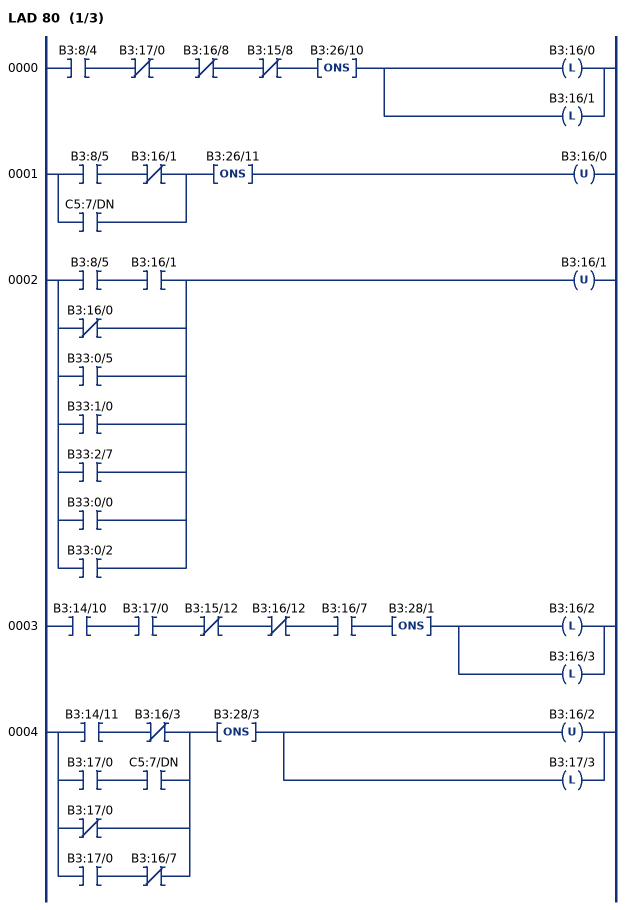
% Rung: 0 %
SOR XIC B3:8/4 XIO B3:17/0 XIO B3:16/8 XIO B3:15/8 OSR B3:26/10 BST OTL B3:16/0 NXB OTL B3:16/1 BND EOR
% Rung: 1 %
SOR BST XIC B3:8/5 XIO B3:16/1 NXB XIC C5:7/DN BND OSR B3:26/11 OTU B3:16/0 EOR
% Rung: 2 %
SOR BST XIC B3:8/5 XIC B3:16/1 NXB XIO B3:16/0 NXB XIC B33:0/5 NXB XIC B33:1/0 NXB XIC B33:2/7 NXB XIC B33:0/0 NXB XIC B33:0/2 BND OTU B3:16/1 EOR
% Rung: 3 %
SOR XIC B3:14/10 XIC B3:17/0 XIO B3:15/12 XIO B3:16/12 XIC B3:16/7 OSR B3:28/1 BST OTL B3:16/2 NXB OTL B3:16/3 BND EOR
% Rung: 4 %
SOR BST XIC B3:14/11 XIO B3:16/3 NXB XIC B3:17/0 XIC C5:7/DN NXB XIO B3:17/0 NXB XIC B3:17/0 XIO B3:16/7 BND OSR B3:28/3 BST OTU B3:16/2 NXB OTL B3:17/3 BND EOR

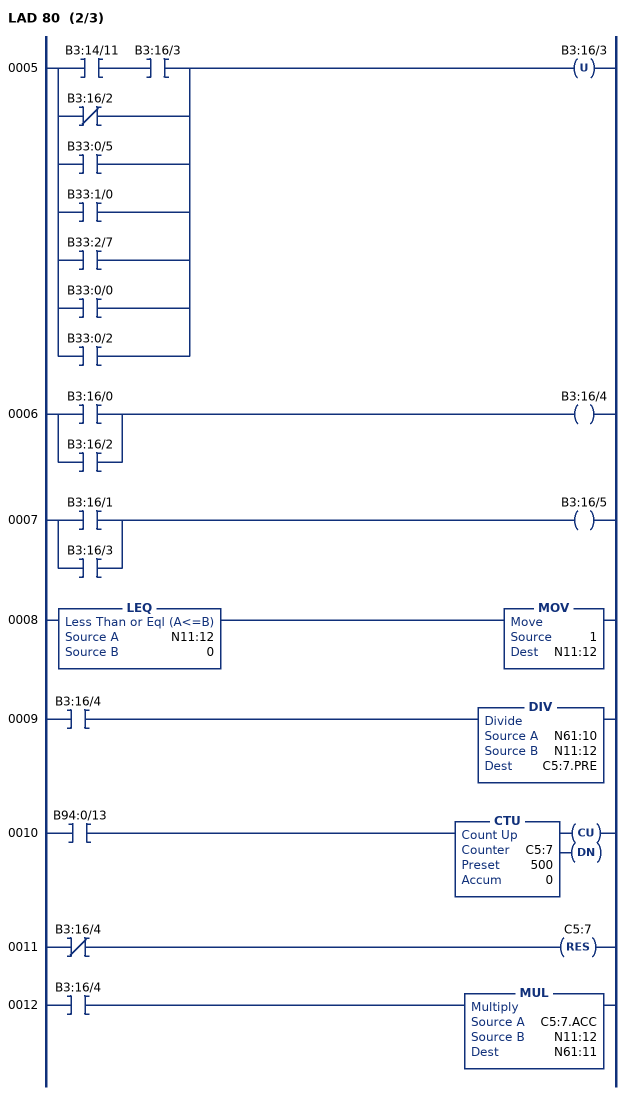
% Rung: 5 %
SOR BST XIC B3:14/11 XIC B3:16/3 NXB XIO B3:16/2 NXB XIC B33:0/5 NXB XIC B33:1/0 NXB XIC B33:2/7 NXB XIC B33:0/0 NXB XIC B33:0/2 BND OTU B3:16/3 EOR
% Rung: 6 %
SOR BST XIC B3:16/0 NXB XIC B3:16/2 BND OTE B3:16/4 EOR
% Rung: 7 %
SOR BST XIC B3:16/1 NXB XIC B3:16/3 BND OTE B3:16/5 EOR
% Rung: 8 %
SOR LEQ N11:12 0 MOV 1 N11:12 EOR
% Rung: 9 %
SOR XIC B3:16/4 DIV N61:10 N11:12 C5:7.PRE EOR
% Rung: 10 %
SOR XIC B94:0/13 CTU C5:7 500 0 EOR
% Rung: 11 %
SOR XIO B3:16/4 RES C5:7 EOR
% Rung: 12 %
SOR XIC B3:16/4 MUL C5:7.ACC N11:12 N61:11 EOR

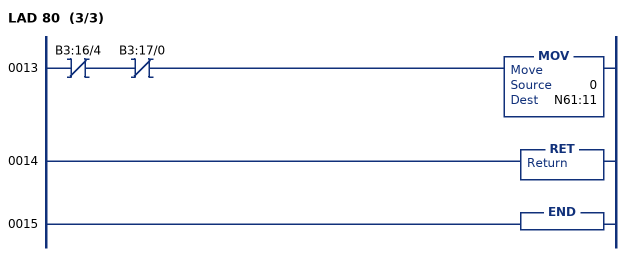
% Rung: 13 %
SOR XIO B3:16/4 XIO B3:17/0 MOV 0 N61:11 EOR
% Rung: 14 %
SOR RET EOR
% Rung: 15 %
SOR END EOR

LADDER 85
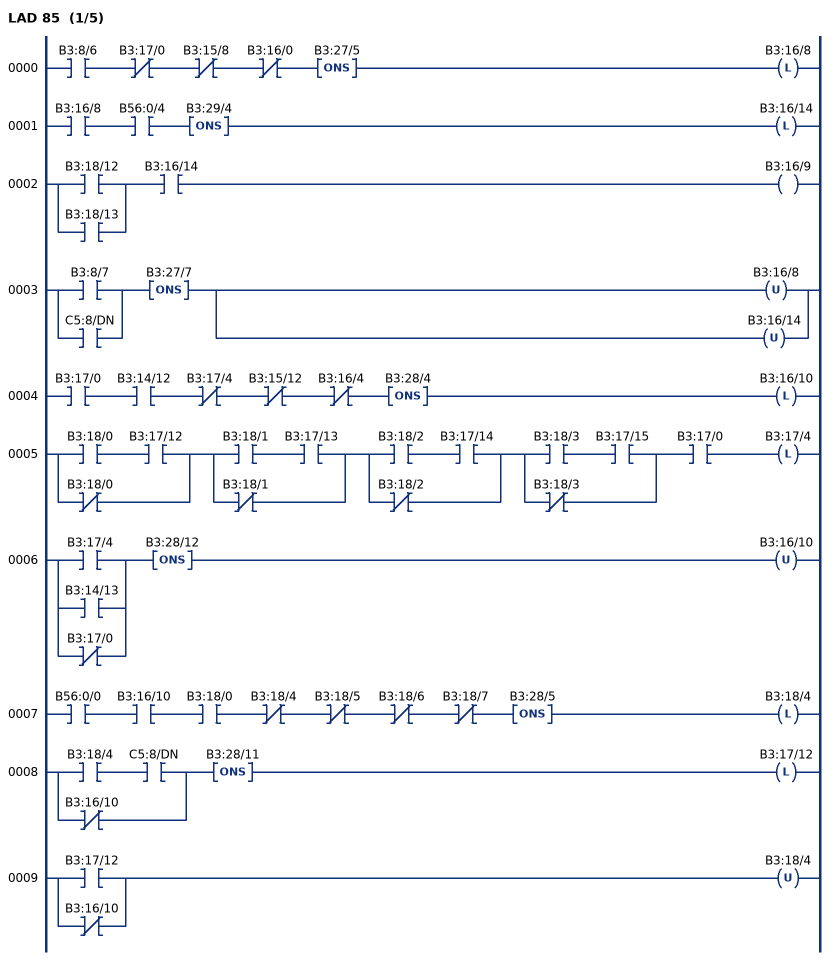
% Rung: 0 %
SOR XIC B3:8/6 XIO B3:17/0 XIO B3:15/8 XIO B3:16/0 OSR B3:27/5 OTL B3:16/8 EOR
% Rung: 1 %
SOR XIC B3:16/8 XIC B56:0/4 OSR B3:29/4 OTL B3:16/14 EOR
% Rung: 2 %
SOR BST XIC B3:18/12 NXB XIC B3:18/13 BND XIC B3:16/14 OTE B3:16/9 EOR
% Rung: 3 %
SOR BST XIC B3:8/7 NXB XIC C5:8/DN BND OSR B3:27/7 BST OTU B3:16/8 NXB OTU B3:16/14 BND EOR
% Rung: 4 %
SOR XIC B3:17/0 XIC B3:14/12 XIO B3:17/4 XIO B3:15/12 XIO B3:16/4 OSR B3:28/4 OTL B3:16/10 EOR
% Rung: 5 %
SOR BST XIC B3:18/0 XIC B3:17/12 NXB XIO B3:18/0 BND BST XIC B3:18/1 XIC B3:17/13 NXB XIO B3:18/1 BND BST XIC B3:18/2 XIC B3:17/14 NXB XIO B3:18/2 BND BST XIC B3:18/3 XIC B3:17/15 NXB XIO B3:18/3 BND XIC B3:17/0 OTL B3:17/4 EOR
% Rung: 6 %
SOR BST XIC B3:17/4 NXB XIC B3:14/13 NXB XIO B3:17/0 BND OSR B3:28/12 OTU B3:16/10 EOR
% Rung: 7 %
SOR XIC B56:0/0 XIC B3:16/10 XIC B3:18/0 XIO B3:18/4 XIO B3:18/5 XIO B3:18/6 XIO B3:18/7 OSR B3:28/5 OTL B3:18/4 EOR
% Rung: 8 %
SOR BST XIC B3:18/4 XIC C5:8/DN NXB XIO B3:16/10 BND OSR B3:28/11 OTL B3:17/12 EOR
% Rung: 9 %
SOR BST XIC B3:17/12 NXB XIO B3:16/10 BND OTU B3:18/4 EOR

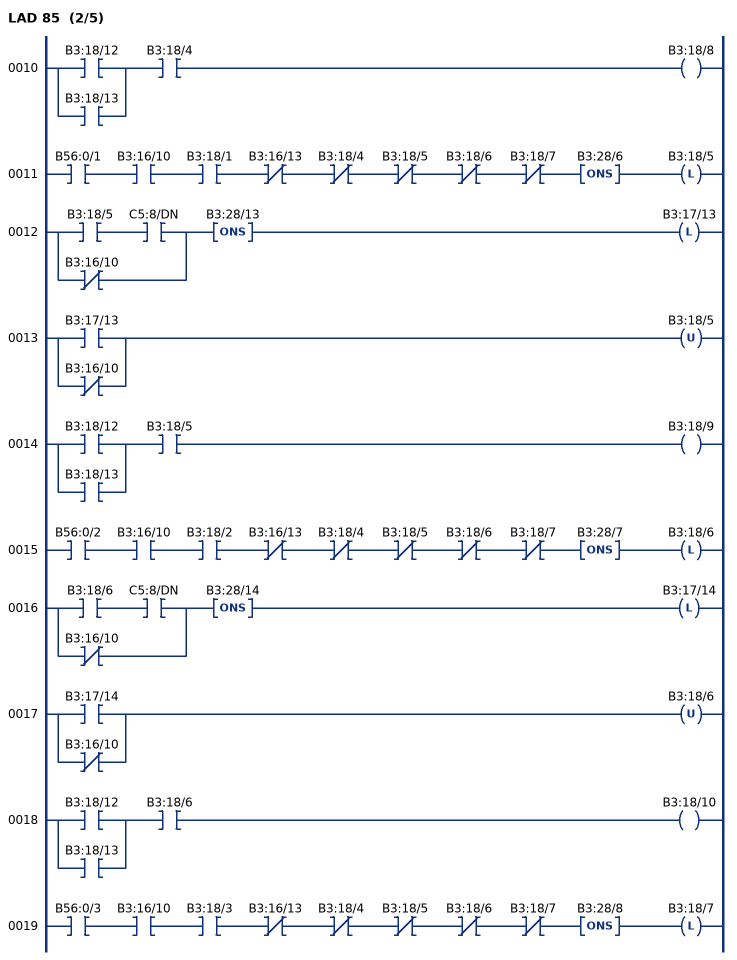
% Rung: 10 %
SOR BST XIC B3:18/12 NXB XIC B3:18/13 BND XIC B3:18/4 OTE B3:18/8 EOR
% Rung: 11 %
SOR XIC B56:0/1 XIC B3:16/10 XIC B3:18/1 XIO B3:16/13 XIO B3:18/4 XIO B3:18/5 XIO B3:18/6 XIO B3:18/7 OSR B3:28/6 OTL B3:18/5 EOR
% Rung: 12 %
SOR BST XIC B3:18/5 XIC C5:8/DN NXB XIO B3:16/10 BND OSR B3:28/13 OTL B3:17/13 EOR
% Rung: 13 %
SOR BST XIC B3:17/13 NXB XIO B3:16/10 BND OTU B3:18/5 EOR
% Rung: 14 %
SOR BST XIC B3:18/12 NXB XIC B3:18/13 BND XIC B3:18/5 OTE B3:18/9 EOR
% Rung: 15 %
SOR XIC B56:0/2 XIC B3:16/10 XIC B3:18/2 XIO B3:16/13 XIO B3:18/4 XIO B3:18/5 XIO B3:18/6 XIO B3:18/7 OSR B3:28/7 OTL B3:18/6 EOR
% Rung: 16 %
SOR BST XIC B3:18/6 XIC C5:8/DN NXB XIO B3:16/10 BND OSR B3:28/14 OTL B3:17/14 EOR
% Rung: 17 %
SOR BST XIC B3:17/14 NXB XIO B3:16/10 BND OTU B3:18/6 EOR
% Rung: 18 %
SOR BST XIC B3:18/12 NXB XIC B3:18/13 BND XIC B3:18/6 OTE B3:18/10 EOR
% Rung: 19 %
SOR XIC B56:0/3 XIC B3:16/10 XIC B3:18/3 XIO B3:16/13 XIO B3:18/4 XIO B3:18/5 XIO B3:18/6 XIO B3:18/7 OSR B3:28/8 OTL B3:18/7 EOR

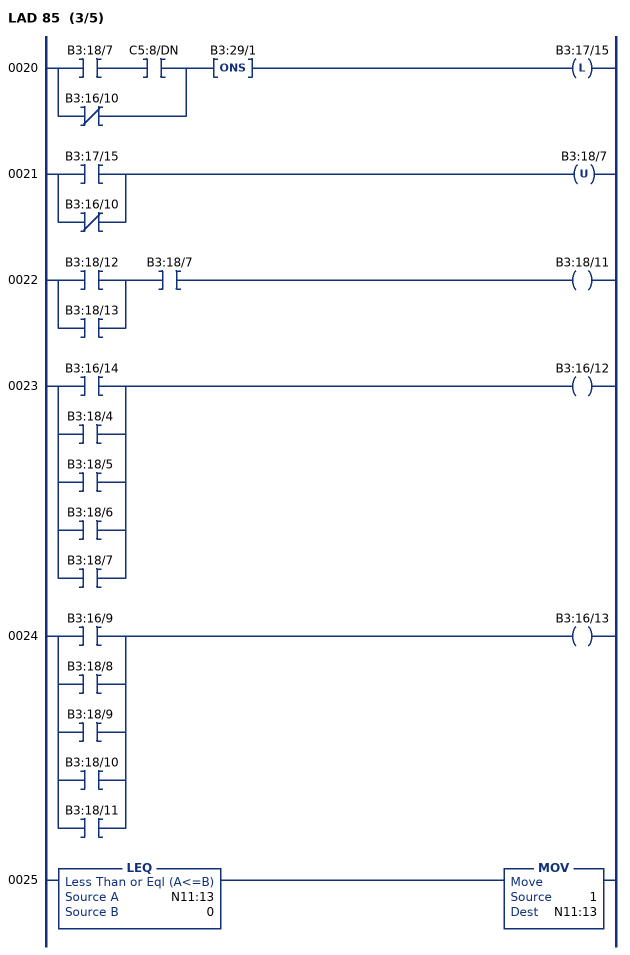
% Rung: 20 %
SOR BST XIC B3:18/7 XIC C5:8/DN NXB XIO B3:16/10 BND OSR B3:29/1 OTL B3:17/15 EOR
% Rung: 21 %
SOR BST XIC B3:17/15 NXB XIO B3:16/10 BND OTU B3:18/7 EOR
% Rung: 22 %
SOR BST XIC B3:18/12 NXB XIC B3:18/13 BND XIC B3:18/7 OTE B3:18/11 EOR
% Rung: 23 %
SOR BST XIC B3:16/14 NXB XIC B3:18/4 NXB XIC B3:18/5 NXB XIC B3:18/6 NXB XIC B3:18/7 BND OTE B3:16/12 EOR
% Rung: 24 %
SOR BST XIC B3:16/9 NXB XIC B3:18/8 NXB XIC B3:18/9 NXB XIC B3:18/10 NXB XIC B3:18/11 BND OTE B3:16/13 EOR
% Rung: 25 %
SOR LEQ N11:13 0 MOV 1 N11:13 EOR

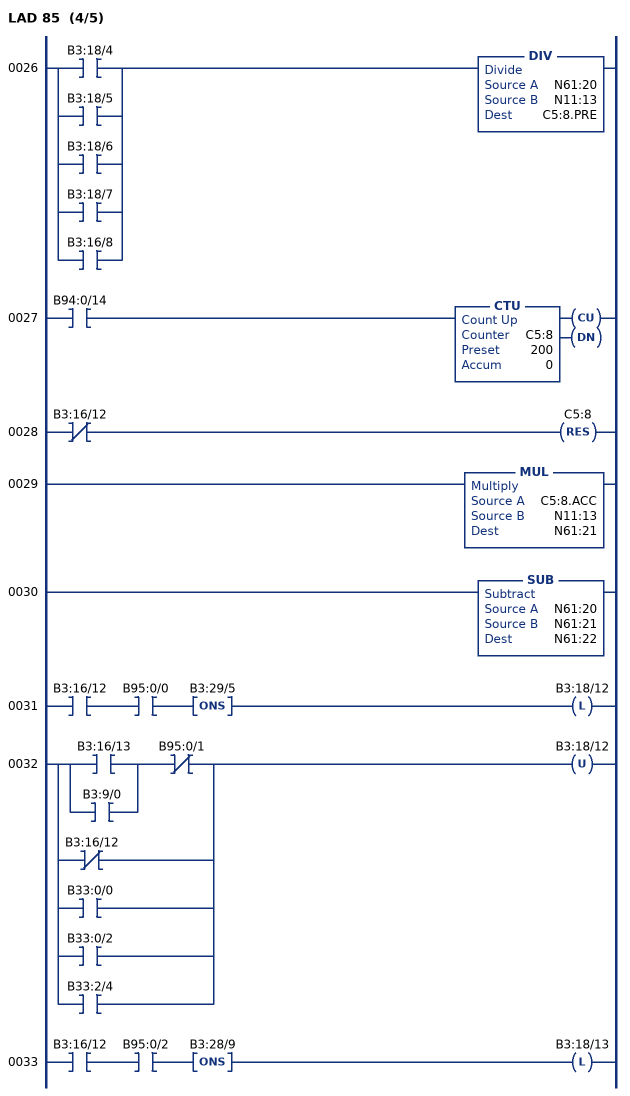
% Rung: 26 %
SOR BST XIC B3:18/4 NXB XIC B3:18/5 NXB XIC B3:18/6 NXB XIC B3:18/7 NXB XIC B3:16/8 BND DIV N61:20 N11:13 C5:8.PRE EOR
% Rung: 27 %
SOR XIC B94:0/14 CTU C5:8 200 0 EOR
% Rung: 28 %
SOR XIO B3:16/12 RES C5:8 EOR
% Rung: 29 %
SOR MUL C5:8.ACC N11:13 N61:21 EOR
% Rung: 30 %
SOR SUB N61:20 N61:21 N61:22 EOR
% Rung: 31 %
SOR XIC B3:16/12 XIC B95:0/0 OSR B3:29/5 OTL B3:18/12 EOR
% Rung: 32 %
SOR BST BST XIC B3:16/13 NXB XIC B3:9/0 BND XIO B95:0/1 NXB XIO B3:16/12 NXB XIC B33:0/0 NXB XIC B33:0/2 NXB XIC B33:2/4 BND OTU B3:18/12 EOR
% Rung: 33 %
SOR XIC B3:16/12 XIC B95:0/2 OSR B3:28/9 OTL B3:18/13 EOR

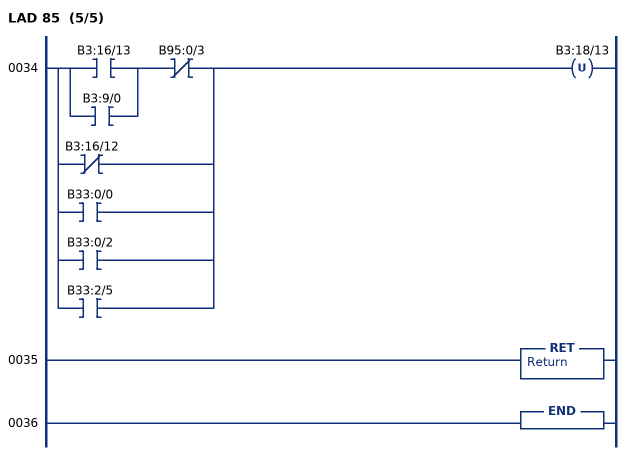
% Rung: 34 %
SOR BST BST XIC B3:16/13 NXB XIC B3:9/0 BND XIO B95:0/3 NXB XIO B3:16/12 NXB XIC B33:0/0 NXB XIC B33:0/2 NXB XIC B33:2/5 BND OTU B3:18/13 EOR
% Rung: 35 %
SOR RET EOR
% Rung: 36 %
SOR END EOR

LADDER 100
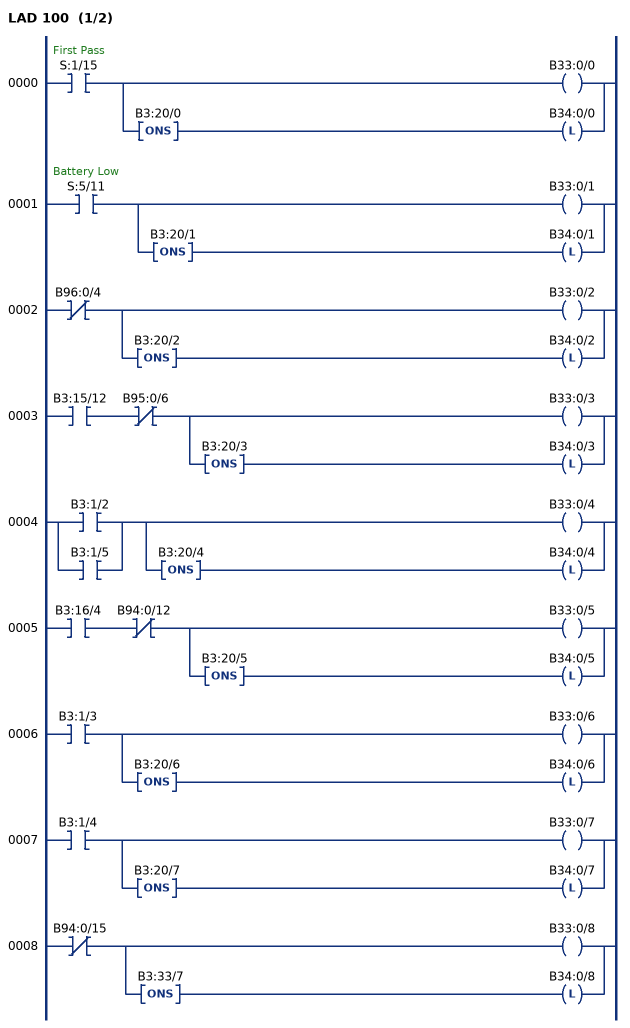
% Rung: 0 %
SOR XIC S:1/15 BST OTE B33:0/0 NXB OSR B3:20/0 OTL B34:0/0 BND EOR
%   S:1/15  "First Pass" %
% Rung: 1 %
SOR XIC S:5/11 BST OTE B33:0/1 NXB OSR B3:20/1 OTL B34:0/1 BND EOR
%   S:5/11  "Battery Low" %
% Rung: 2 %
SOR XIO B96:0/4 BST OTE B33:0/2 NXB OSR B3:20/2 OTL B34:0/2 BND EOR
% Rung: 3 %
SOR XIC B3:15/12 XIO B95:0/6 BST OTE B33:0/3 NXB OSR B3:20/3 OTL B34:0/3 BND EOR
% Rung: 4 %
SOR BST XIC B3:1/2 NXB XIC B3:1/5 BND BST OTE B33:0/4 NXB OSR B3:20/4 OTL B34:0/4 BND EOR
% Rung: 5 %
SOR XIC B3:16/4 XIO B94:0/12 BST OTE B33:0/5 NXB OSR B3:20/5 OTL B34:0/5 BND EOR
% Rung: 6 %
SOR XIC B3:1/3 BST OTE B33:0/6 NXB OSR B3:20/6 OTL B34:0/6 BND EOR
% Rung: 7 %
SOR XIC B3:1/4 BST OTE B33:0/7 NXB OSR B3:20/7 OTL B34:0/7 BND EOR
% Rung: 8 %
SOR XIO B94:0/15 BST OTE B33:0/8 NXB OSR B3:33/7 OTL B34:0/8 BND EOR

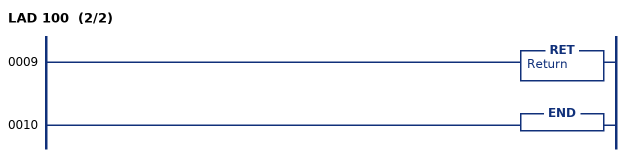
% Rung: 9 %
SOR RET EOR
% Rung: 10 %
SOR END EOR

LADDER 101
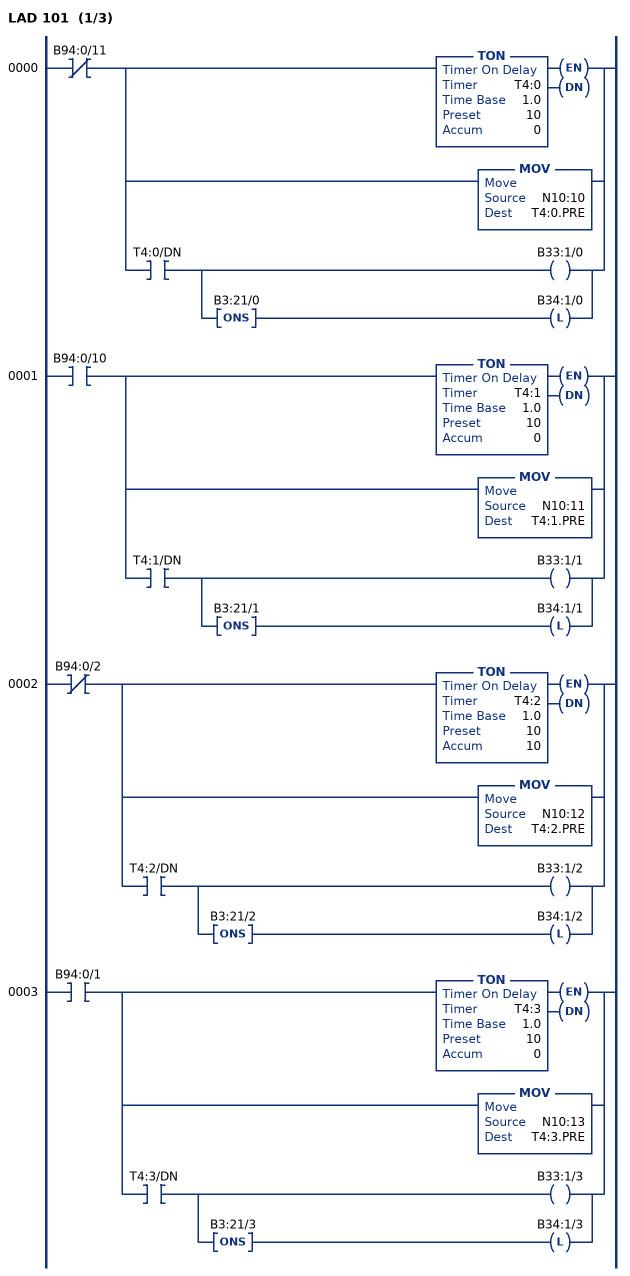
% Rung: 0 %
SOR XIO B94:0/11 BST TON T4:0 1.0 10 0 NXB MOV N10:10 T4:0.PRE NXB XIC T4:0/DN BST OTE B33:1/0 NXB OSR B3:21/0 OTL B34:1/0 BND BND EOR
% Rung: 1 %
SOR XIC B94:0/10 BST TON T4:1 1.0 10 0 NXB MOV N10:11 T4:1.PRE NXB XIC T4:1/DN BST OTE B33:1/1 NXB OSR B3:21/1 OTL B34:1/1 BND BND EOR
% Rung: 2 %
SOR XIO B94:0/2 BST TON T4:2 1.0 10 10 NXB MOV N10:12 T4:2.PRE NXB XIC T4:2/DN BST OTE B33:1/2 NXB OSR B3:21/2 OTL B34:1/2 BND BND EOR
% Rung: 3 %
SOR XIC B94:0/1 BST TON T4:3 1.0 10 0 NXB MOV N10:13 T4:3.PRE NXB XIC T4:3/DN BST OTE B33:1/3 NXB OSR B3:21/3 OTL B34:1/3 BND BND EOR

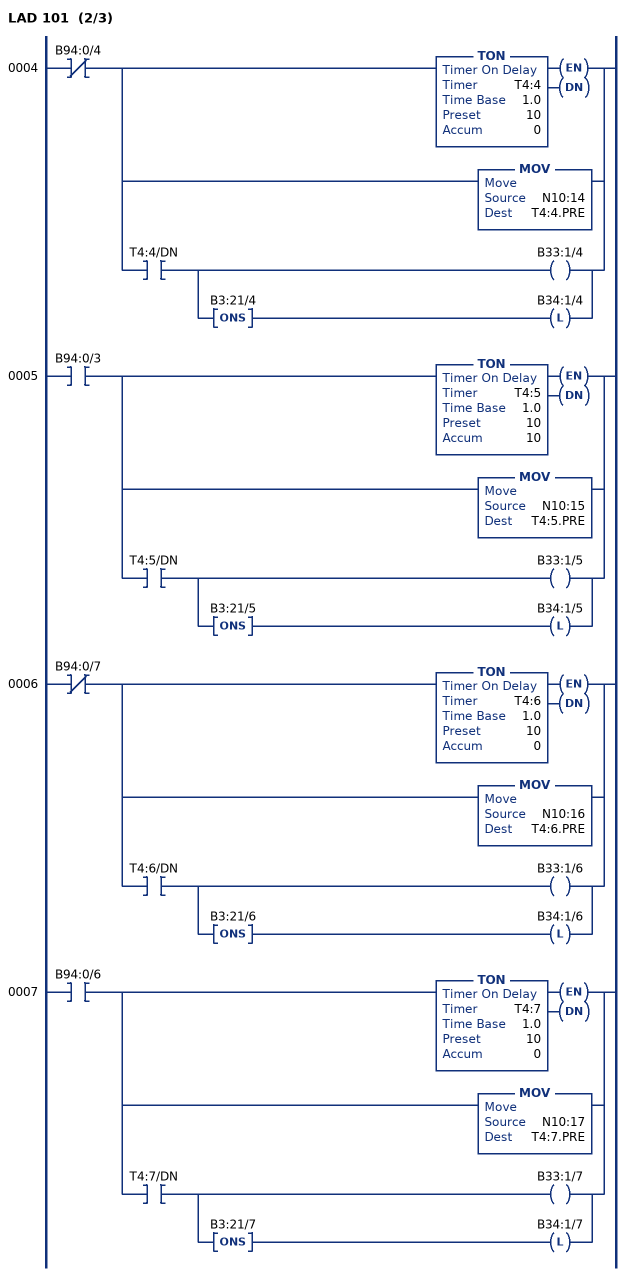
% Rung: 4 %
SOR XIO B94:0/4 BST TON T4:4 1.0 10 0 NXB MOV N10:14 T4:4.PRE NXB XIC T4:4/DN BST OTE B33:1/4 NXB OSR B3:21/4 OTL B34:1/4 BND BND EOR
% Rung: 5 %
SOR XIC B94:0/3 BST TON T4:5 1.0 10 10 NXB MOV N10:15 T4:5.PRE NXB XIC T4:5/DN BST OTE B33:1/5 NXB OSR B3:21/5 OTL B34:1/5 BND BND EOR
% Rung: 6 %
SOR XIO B94:0/7 BST TON T4:6 1.0 10 0 NXB MOV N10:16 T4:6.PRE NXB XIC T4:6/DN BST OTE B33:1/6 NXB OSR B3:21/6 OTL B34:1/6 BND BND EOR
% Rung: 7 %
SOR XIC B94:0/6 BST TON T4:7 1.0 10 0 NXB MOV N10:17 T4:7.PRE NXB XIC T4:7/DN BST OTE B33:1/7 NXB OSR B3:21/7 OTL B34:1/7 BND BND EOR

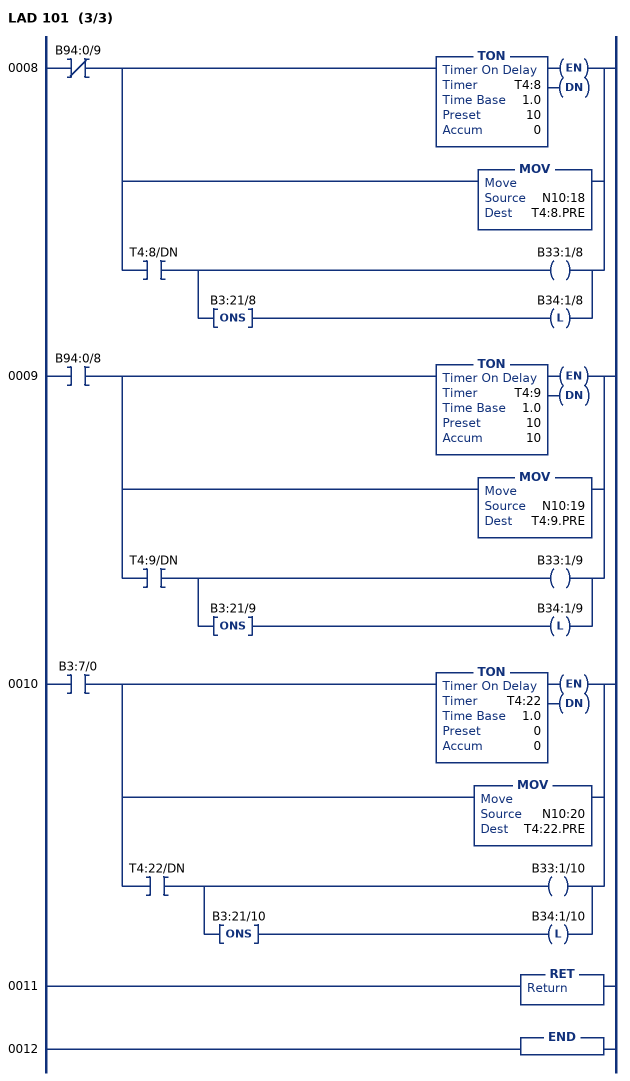
% Rung: 8 %
SOR XIO B94:0/9 BST TON T4:8 1.0 10 0 NXB MOV N10:18 T4:8.PRE NXB XIC T4:8/DN BST OTE B33:1/8 NXB OSR B3:21/8 OTL B34:1/8 BND BND EOR
% Rung: 9 %
SOR XIC B94:0/8 BST TON T4:9 1.0 10 10 NXB MOV N10:19 T4:9.PRE NXB XIC T4:9/DN BST OTE B33:1/9 NXB OSR B3:21/9 OTL B34:1/9 BND BND EOR
% Rung: 10 %
SOR XIC B3:7/0 BST TON T4:22 1.0 0 0 NXB MOV N10:20 T4:22.PRE NXB XIC T4:22/DN BST OTE B33:1/10 NXB OSR B3:21/10 OTL B34:1/10 BND BND EOR
% Rung: 11 %
SOR RET EOR
% Rung: 12 %
SOR END EOR

LADDER 102
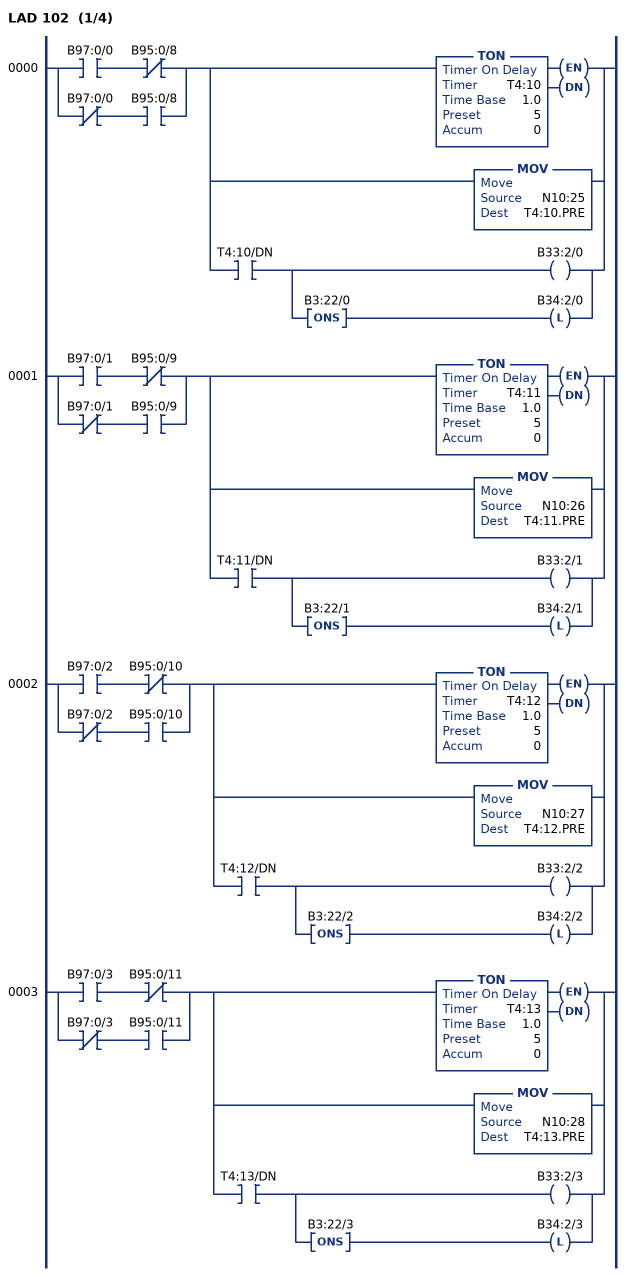
% Rung: 0 %
SOR BST XIC B97:0/0 XIO B95:0/8 NXB XIO B97:0/0 XIC B95:0/8 BND BST TON T4:10 1.0 5 0 NXB MOV N10:25 T4:10.PRE NXB XIC T4:10/DN BST OTE B33:2/0 NXB OSR B3:22/0 OTL B34:2/0 BND BND EOR
% Rung: 1 %
SOR BST XIC B97:0/1 XIO B95:0/9 NXB XIO B97:0/1 XIC B95:0/9 BND BST TON T4:11 1.0 5 0 NXB MOV N10:26 T4:11.PRE NXB XIC T4:11/DN BST OTE B33:2/1 NXB OSR B3:22/1 OTL B34:2/1 BND BND EOR
% Rung: 2 %
SOR BST XIC B97:0/2 XIO B95:0/10 NXB XIO B97:0/2 XIC B95:0/10 BND BST TON T4:12 1.0 5 0 NXB MOV N10:27 T4:12.PRE NXB XIC T4:12/DN BST OTE B33:2/2 NXB OSR B3:22/2 OTL B34:2/2 BND BND EOR
% Rung: 3 %
SOR BST XIC B97:0/3 XIO B95:0/11 NXB XIO B97:0/3 XIC B95:0/11 BND BST TON T4:13 1.0 5 0 NXB MOV N10:28 T4:13.PRE NXB XIC T4:13/DN BST OTE B33:2/3 NXB OSR B3:22/3 OTL B34:2/3 BND BND EOR

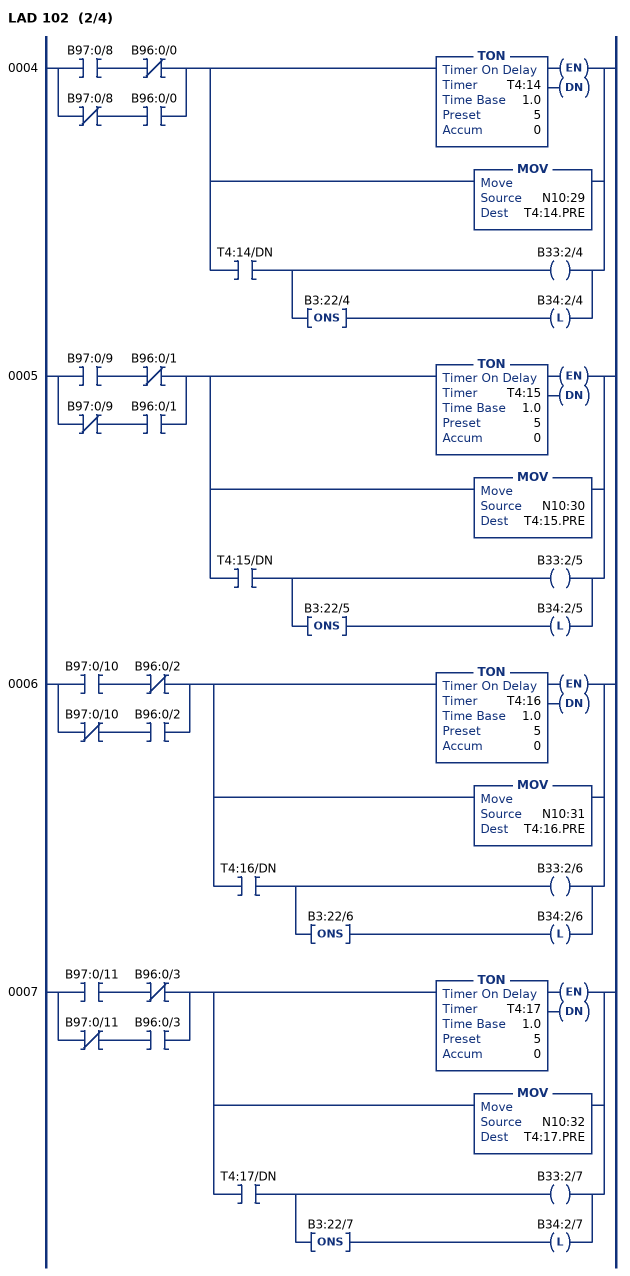
% Rung: 4 %
SOR BST XIC B97:0/8 XIO B96:0/0 NXB XIO B97:0/8 XIC B96:0/0 BND BST TON T4:14 1.0 5 0 NXB MOV N10:29 T4:14.PRE NXB XIC T4:14/DN BST OTE B33:2/4 NXB OSR B3:22/4 OTL B34:2/4 BND BND EOR
% Rung: 5 %
SOR BST XIC B97:0/9 XIO B96:0/1 NXB XIO B97:0/9 XIC B96:0/1 BND BST TON T4:15 1.0 5 0 NXB MOV N10:30 T4:15.PRE NXB XIC T4:15/DN BST OTE B33:2/5 NXB OSR B3:22/5 OTL B34:2/5 BND BND EOR
% Rung: 6 %
SOR BST XIC B97:0/10 XIO B96:0/2 NXB XIO B97:0/10 XIC B96:0/2 BND BST TON T4:16 1.0 5 0 NXB MOV N10:31 T4:16.PRE NXB XIC T4:16/DN BST OTE B33:2/6 NXB OSR B3:22/6 OTL B34:2/6 BND BND EOR
% Rung: 7 %
SOR BST XIC B97:0/11 XIO B96:0/3 NXB XIO B97:0/11 XIC B96:0/3 BND BST TON T4:17 1.0 5 0 NXB MOV N10:32 T4:17.PRE NXB XIC T4:17/DN BST OTE B33:2/7 NXB OSR B3:22/7 OTL B34:2/7 BND BND EOR

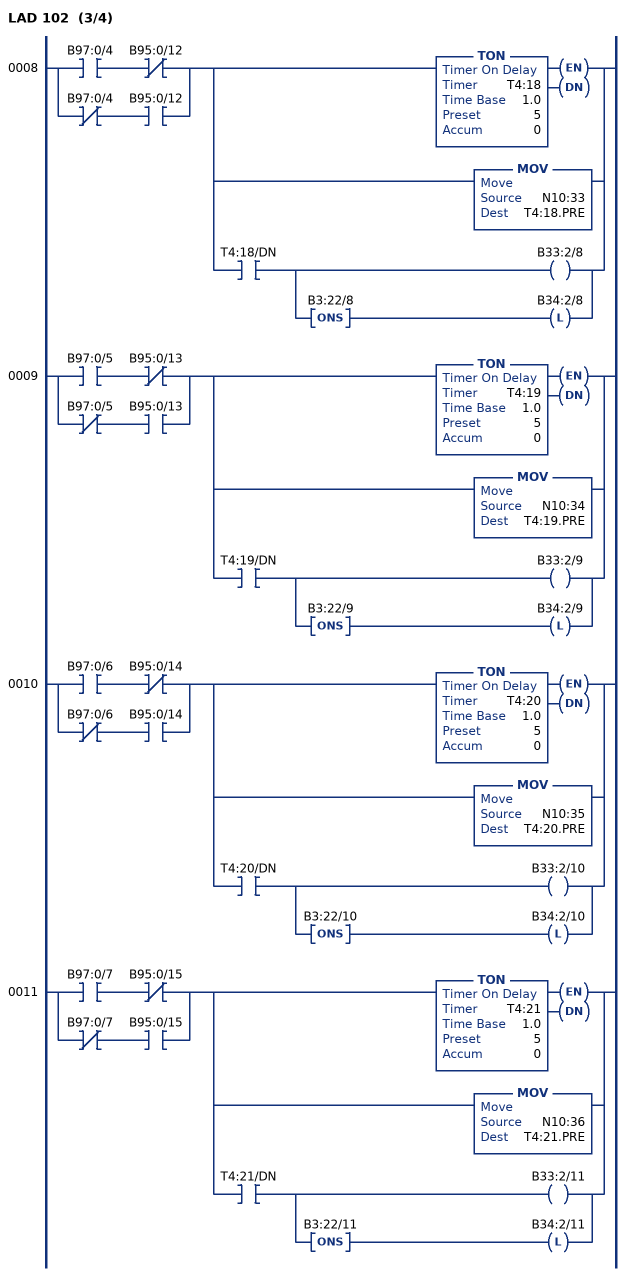
% Rung: 8 %
SOR BST XIC B97:0/4 XIO B95:0/12 NXB XIO B97:0/4 XIC B95:0/12 BND BST TON T4:18 1.0 5 0 NXB MOV N10:33 T4:18.PRE NXB XIC T4:18/DN BST OTE B33:2/8 NXB OSR B3:22/8 OTL B34:2/8 BND BND EOR
% Rung: 9 %
SOR BST XIC B97:0/5 XIO B95:0/13 NXB XIO B97:0/5 XIC B95:0/13 BND BST TON T4:19 1.0 5 0 NXB MOV N10:34 T4:19.PRE NXB XIC T4:19/DN BST OTE B33:2/9 NXB OSR B3:22/9 OTL B34:2/9 BND BND EOR
% Rung: 10 %
SOR BST XIC B97:0/6 XIO B95:0/14 NXB XIO B97:0/6 XIC B95:0/14 BND BST TON T4:20 1.0 5 0 NXB MOV N10:35 T4:20.PRE NXB XIC T4:20/DN BST OTE B33:2/10 NXB OSR B3:22/10 OTL B34:2/10 BND BND EOR
% Rung: 11 %
SOR BST XIC B97:0/7 XIO B95:0/15 NXB XIO B97:0/7 XIC B95:0/15 BND BST TON T4:21 1.0 5 0 NXB MOV N10:36 T4:21.PRE NXB XIC T4:21/DN BST OTE B33:2/11 NXB OSR B3:22/11 OTL B34:2/11 BND BND EOR

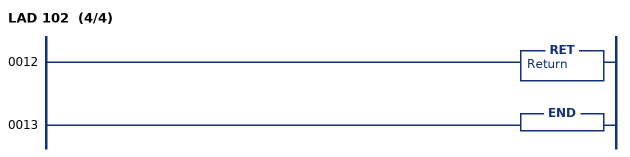
% Rung: 12 %
SOR RET EOR
% Rung: 13 %
SOR END EOR

LADDER 103
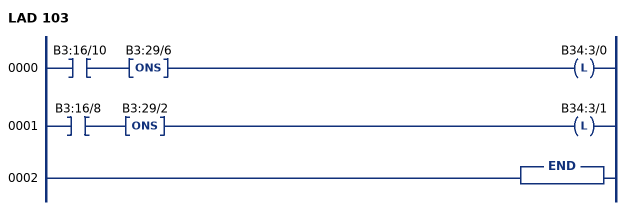
% Rung: 0 %
SOR XIC B3:16/10 OSR B3:29/6 OTL B34:3/0 EOR
% Rung: 1 %
SOR XIC B3:16/8 OSR B3:29/2 OTL B34:3/1 EOR
% Rung: 2 %
SOR END EOR

LADDER 110
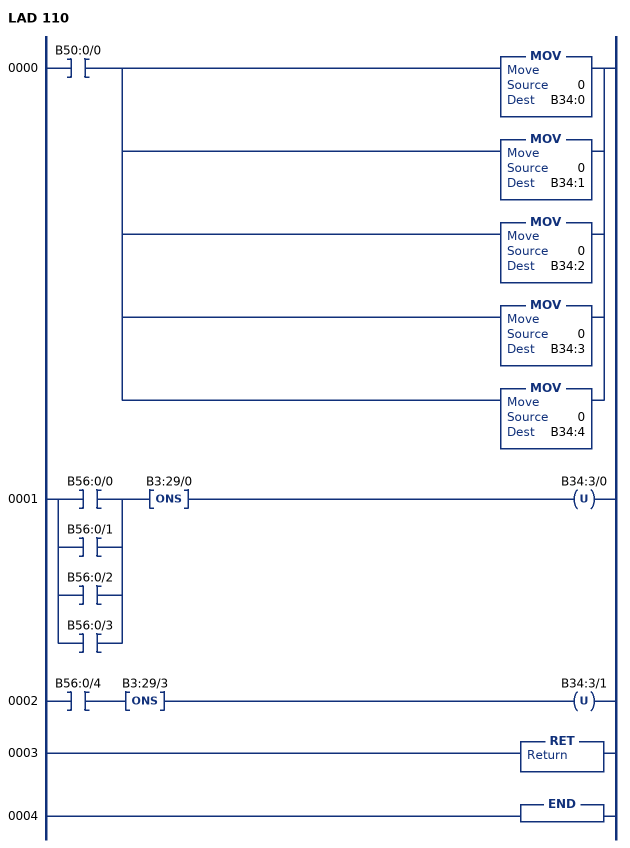
% Rung: 0 %
SOR XIC B50:0/0 BST MOV 0 B34:0 NXB MOV 0 B34:1 NXB MOV 0 B34:2 NXB MOV 0 B34:3 NXB MOV 0 B34:4 BND EOR
% Rung: 1 %
SOR BST XIC B56:0/0 NXB XIC B56:0/1 NXB XIC B56:0/2 NXB XIC B56:0/3 BND OSR B3:29/0 OTU B34:3/0 EOR
% Rung: 2 %
SOR XIC B56:0/4 OSR B3:29/3 OTU B34:3/1 EOR
% Rung: 3 %
SOR RET EOR
% Rung: 4 %
SOR END EOR

LADDER 200
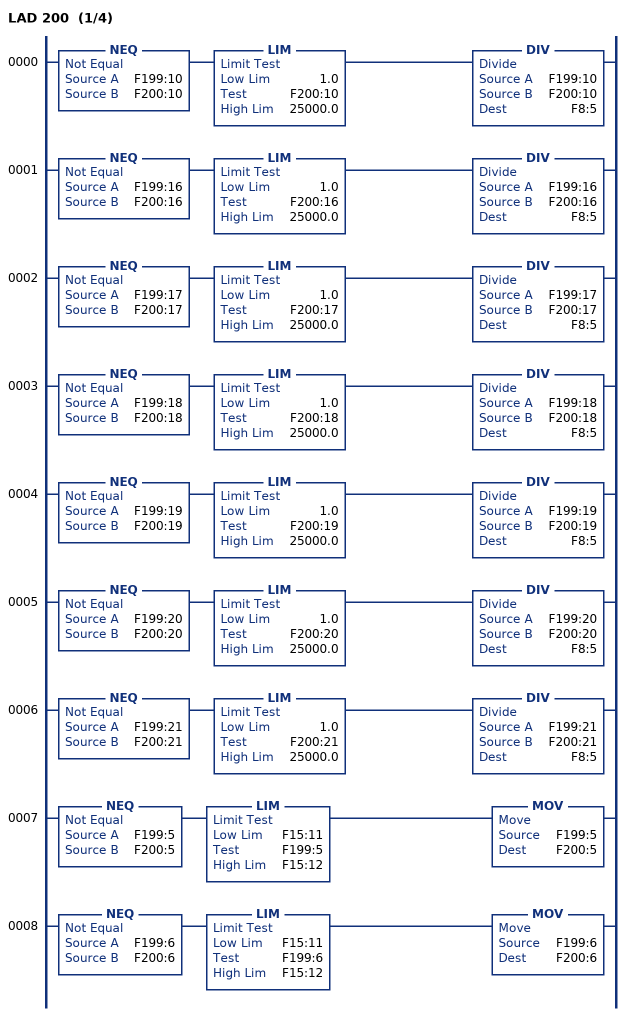
% Rung: 0 %
SOR NEQ F199:10 F200:10 LIM 1.0 F200:10 25000.0 DIV F199:10 F200:10 F8:5 EOR
% Rung: 1 %
SOR NEQ F199:16 F200:16 LIM 1.0 F200:16 25000.0 DIV F199:16 F200:16 F8:5 EOR
% Rung: 2 %
SOR NEQ F199:17 F200:17 LIM 1.0 F200:17 25000.0 DIV F199:17 F200:17 F8:5 EOR
% Rung: 3 %
SOR NEQ F199:18 F200:18 LIM 1.0 F200:18 25000.0 DIV F199:18 F200:18 F8:5 EOR
% Rung: 4 %
SOR NEQ F199:19 F200:19 LIM 1.0 F200:19 25000.0 DIV F199:19 F200:19 F8:5 EOR
% Rung: 5 %
SOR NEQ F199:20 F200:20 LIM 1.0 F200:20 25000.0 DIV F199:20 F200:20 F8:5 EOR
% Rung: 6 %
SOR NEQ F199:21 F200:21 LIM 1.0 F200:21 25000.0 DIV F199:21 F200:21 F8:5 EOR
% Rung: 7 %
SOR NEQ F199:5 F200:5 LIM F15:11 F199:5 F15:12 MOV F199:5 F200:5 EOR
% Rung: 8 %
SOR NEQ F199:6 F200:6 LIM F15:11 F199:6 F15:12 MOV F199:6 F200:6 EOR

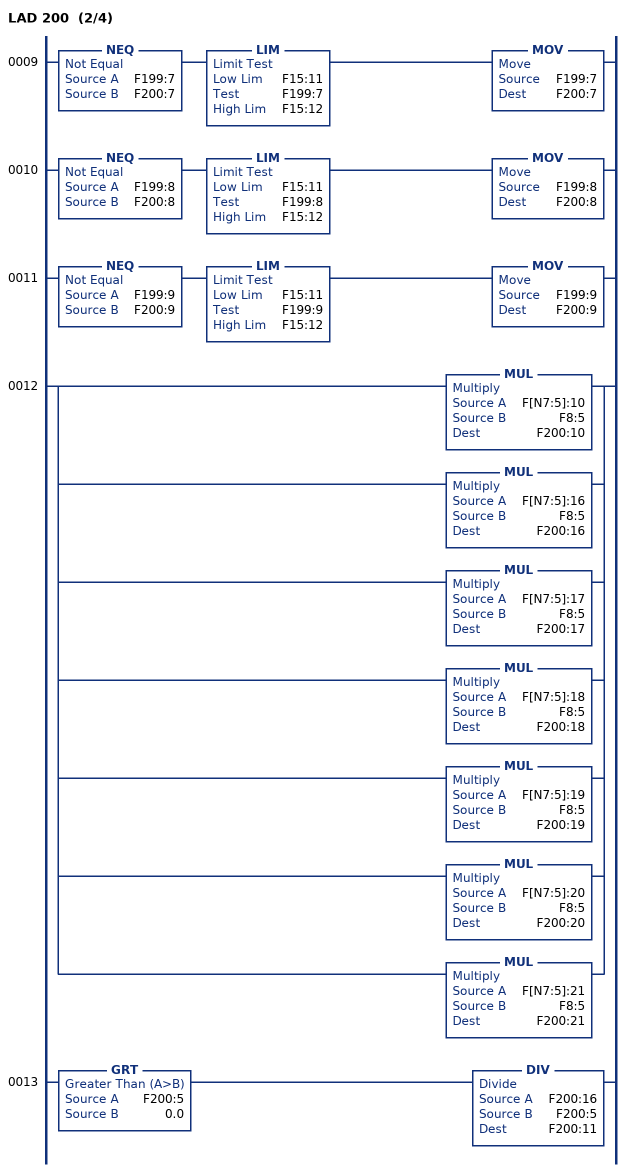
% Rung: 9 %
SOR NEQ F199:7 F200:7 LIM F15:11 F199:7 F15:12 MOV F199:7 F200:7 EOR
% Rung: 10 %
SOR NEQ F199:8 F200:8 LIM F15:11 F199:8 F15:12 MOV F199:8 F200:8 EOR
% Rung: 11 %
SOR NEQ F199:9 F200:9 LIM F15:11 F199:9 F15:12 MOV F199:9 F200:9 EOR
% Rung: 12 %
SOR BST MUL F[N7:5]:10 F8:5 F200:10 NXB MUL F[N7:5]:16 F8:5 F200:16 NXB MUL F[N7:5]:17 F8:5 F200:17 NXB MUL F[N7:5]:18 F8:5 F200:18 NXB MUL F[N7:5]:19 F8:5 F200:19 NXB MUL F[N7:5]:20 F8:5 F200:20 NXB MUL F[N7:5]:21 F8:5 F200:21 BND EOR
% Rung: 13 %
SOR GRT F200:5 0.0 DIV F200:16 F200:5 F200:11 EOR

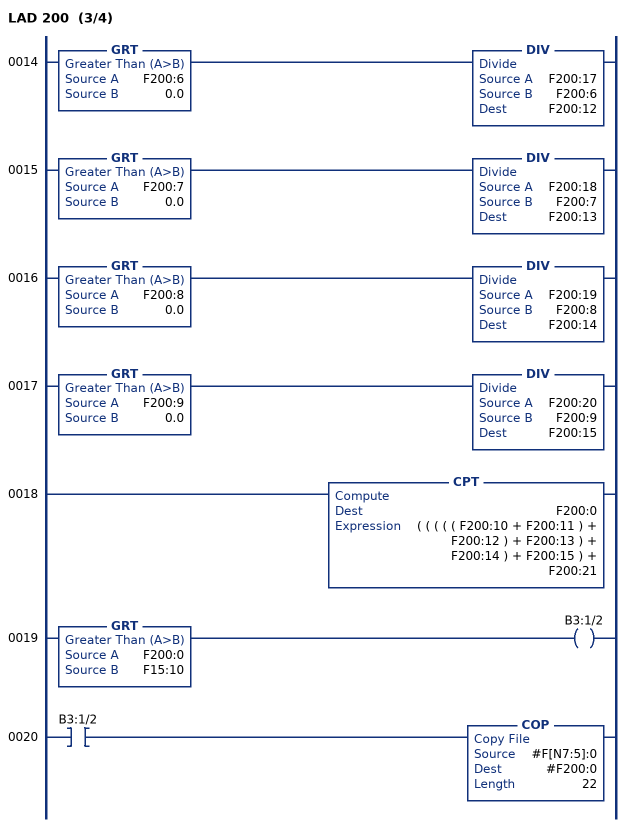
% Rung: 14 %
SOR GRT F200:6 0.0 DIV F200:17 F200:6 F200:12 EOR
% Rung: 15 %
SOR GRT F200:7 0.0 DIV F200:18 F200:7 F200:13 EOR
% Rung: 16 %
SOR GRT F200:8 0.0 DIV F200:19 F200:8 F200:14 EOR
% Rung: 17 %
SOR GRT F200:9 0.0 DIV F200:20 F200:9 F200:15 EOR
% Rung: 18 %
SOR CPT F200:0 " ( ( ( ( ( F200:10 + F200:11 ) + F200:12 ) + F200:13 ) + F200:14 ) + F200:15 ) + F200:21 " EOR
% Rung: 19 %
SOR GRT F200:0 F15:10 OTE B3:1/2 EOR
% Rung: 20 %
SOR XIC B3:1/2 COP #F[N7:5]:0 #F200:0 22 EOR

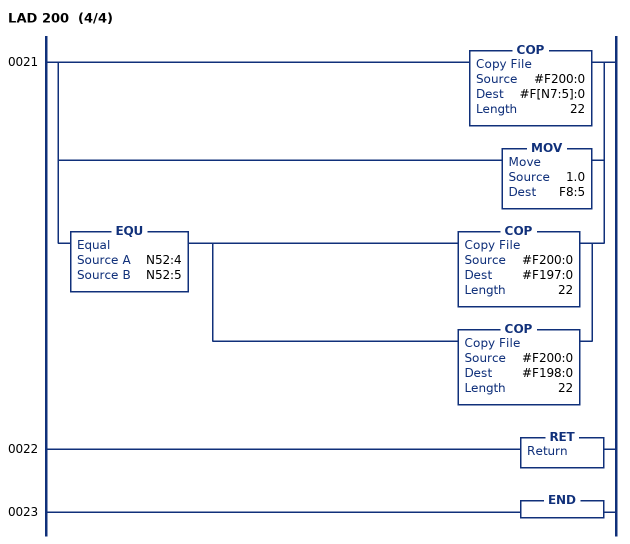
% Rung: 21 %
SOR BST BST COP #F200:0 #F[N7:5]:0 22 NXB MOV 1.0 F8:5 BND NXB EQU N52:4 N52:5 BST COP #F200:0 #F197:0 22 NXB COP #F200:0 #F198:0 22 BND BND EOR
% Rung: 22 %
SOR RET EOR
% Rung: 23 %
SOR END EOR

DATA TABLE (non-zero values as saved)
DATA B3
% B3:0 % 0X0006 0X0000 0X0000 0X0000 0X0000 0X0000 0X0000 0X0000 0X0000 0X0000
% B3:10 % 0X0020 0X0000 0X5100 0X0400 0X0000 0X0000 0X0000 0X0003 0X0001 0X0000
% B3:20 % 0X0000 0X0224 0X0000 0X0000 0X0000 0X2000 0X7020 0XB840 0X6C0D 0X0002
% B3:40 % 0X0001 0X0000 0X0000 0X0000 0X0000 0X0000 0X0000 0X0000 0X0000 0X0000
% B3:70 % 0X0001 0X0000 0X0000 0X0000 0X0000 0X0000 0X0000 0X0000 0X0000 0X0000
DATA T4
% .PRE .ACC %
% T4:0 % 10 0
% T4:1 % 10 0
% T4:2 % 10 10
% T4:3 % 10 0
% T4:4 % 10 0
% T4:5 % 10 10
% T4:6 % 10 0
% T4:7 % 10 0
% T4:8 % 10 0
% T4:9 % 10 10
% T4:10 % 5 0
% T4:11 % 5 0
% T4:12 % 5 0
% T4:13 % 5 0
% T4:14 % 5 0
% T4:15 % 5 0
% T4:16 % 5 0
% T4:17 % 5 0
% T4:18 % 5 0
% T4:19 % 5 0
% T4:20 % 5 0
% T4:21 % 5 0
% T4:26 % 300 88
% T4:28 % 300 158
% T4:30 % 80 6
% T4:31 % 80 0
% T4:32 % 1 0
% T4:33 % 1 0
% T4:40 % 1 0
% T4:42 % 5 5
% T4:43 % 5 0
% T4:44 % 5 5
% T4:45 % 5 5
% T4:52 % 3 0
% T4:80 % 1 0
% T4:84 % 5 0
% T4:87 % 5 0
% T4:88 % 5 0
% T4:89 % 30 0
% T4:90 % 5 0
DATA C5
% .PRE .ACC %
% C5:5 % 80 0
% C5:6 % 10 0
% C5:7 % 500 0
% C5:8 % 200 0
DATA N7
% N7:0 % 0 0 0 1 1 201 0 0 0 0
% N7:10 % 1 1 201 0 0 0 0 0 0 0
% N7:30 % 10 99 15 3 0 0 0 0 0 0
% N7:40 % 10 11 0 99 15 15 0 19 0 0
% N7:70 % 0 10 10 10 10 60 0 0 0 0
% N7:80 % 2419 0 89 299 0 70 50 50 700 700
% N7:90 % -28 0 30 100 0 8630 9950 9950 24300 24300
% N7:100 % 2329 1 1 1 1 0 0 0 5000 5000
DATA F8
% F8:0 % 90 95 85 0 0
% F8:5 % 1 0 0 0 0
DATA N10
% N10:0 % 1023 0 1 0 0 0 0 0 0 0
% N10:10 % 10 10 10 10 10 10 10 10 10 10
% N10:20 % 0 0 0 0 0 5 5 5 5 5
% N10:30 % 5 5 5 5 5 5 5 0 0 0
% N10:50 % 5 30 5 5 5 0 0 0 0 0
% N10:60 % 8700 10000 10000 25000 25000 0 0 0 0 0
% N10:70 % 10 10 10 10 10 2 2 2 2 2
% N10:80 % 98 150 150 2100 2100 0 0 0 0 0
% N10:90 % 300 0 300 0 0 0 1500 1000 23000 20000
DATA N11
% N11:0 % 1 50 0 0 0 0 0 0 0 0
% N11:10 % 10 10 10 10 0 0 0 0 0 0
% N11:70 % 1 0 0 0 50 30 0 100 0 100
% N11:80 % 0 10 10 10 10 60 0 0 0 0
DATA F15
% F15:0 % 2 7 0.01 90 90
% F15:5 % 5 5 0 0 0
% F15:10 % 25000 0.001 10 0 0
DATA N20
% N20:0 % 18 0 9830 200 700 1 0 16383 0 0
% N20:10 % 0 16383 0 10 0 0 0 0 0 0
% N20:20 % 0 0 0 16383 16383 0 0 0 0 0
DATA N30
% N30:60 % 97 7 0 7 17 0 0 0 0 0
DATA B33
% B33:0 % 0X0000 0X0224 0X0000 0X0000 0X0000
DATA B34
% B34:0 % 0X0000 0X008C 0X01C0 0X0000 0X0000
DATA B51
% B51:0 % 0X0000 0X0000 0X0000 0X0000 0X0000 0X0224 0X0000 0X0000 0X0000 0X0000
% B51:20 % 0X0000 0X1000 0X0000 0X0000 0X0000 0X0000 0X0000 0X0000 0X0000 0X0000
% B51:30 % 0X0000 0X02AC 0X01C0 0X0000 0X0000 0X0000 0X0000 0X0000 0X0000 0X0000
DATA N52
% N52:0 % 0 7 0 0 1 1 0 0 0 0
% N52:10 % 0 1 0 0 0 0 0 0 0 0
% N52:20 % 5000 2300 0 500 50 30 0 0 0 0
% N52:30 % 10 99 15 3 20000 0 0 0 0 0
% N52:40 % 1 1 0 0 0 0 0 0 14 16
% N52:60 % 2002 1 22 23 51 45 0 0 0 0
DATA N53
% N53:0 % 1 2 1 1 0 0 0 0 20000 0
% N53:10 % 0 0 0 0 0 0 2 0 2 2
% N53:20 % 0 0 0 0 0 0 0 0 0 2
% N53:30 % 23010 1 31 99 1 0 0 0 0 0
% N53:40 % 0 0 16 17 0 2 0 0 0 0
% N53:50 % 800 800 0 0 0 0 160 0 0 0
% N53:60 % 23 7 12 17 21 33 0 0 0 0
DATA F54
% F54:0 % 2 7 0.01 90 100
% F54:5 % 90 0 0 0 0
DATA F55
% F55:0 % 150 90 0 25.85607 150
% F55:5 % 90 0 0 0 0
DATA N58
% N58:0 % 2 0 0 0 0 0 0 0 0 0
% N58:10 % 0 0 0 0 0 0 16 17 0 0
DATA N59
% N59:0 % -32768 0 0 0 0 0 0 0 0 0
% N59:20 % 8192 2 1 54 137 60 0 224 5 245
% N59:30 % 0 2 3072 0 0 0 0 0 0 0
% N59:40 % 0 0 256 256 256 256 0 0 0 0
% N59:60 % 8192 3 4 231 137 42 0 160 5 245
% N59:70 % 0 8 3072 0 0 0 0 0 0 0
% N59:80 % 8192 3 4 231 137 2 0 96 5 245
% N59:90 % 0 8 3072 0 0 0 256 0 0 0
% N59:100 % 8192 3 1 232 137 41 0 32 5 245
% N59:110 % 0 2 3072 0 0 0 129 0 0 0
% N59:120 % -32768 3 1 232 137 1 0 228 5 246
% N59:130 % 0 2 4096 0
DATA N60
% N60:0 % 264 0 0 0 0 0 12 12 12 12
% N60:10 % 0 8 8 8 8
DATA N61
% N61:0 % 800 800 0 0 0 0 0 0 0 0
% N61:20 % 2000 0 2000 0 0 0 0 0 0 0
DATA B94
% B94:0 % 0X8B98
DATA B95
% B95:0 % 0X000A
DATA B96
% B96:0 % 0X0010
DATA B98
% B98:0 % 0X1000
DATA B99
% B99:0 % 0X1100
DATA F197
% F197:0 % 959.9999 0 0 16 17
% F197:5 % 1 1 1 1 1.001
% F197:10 % 800 0 0 160 0
% F197:15 % 0 0 0 160 0
DATA F198
% F198:0 % 959.9999 0 0 16 17
% F198:5 % 1 1 1 1 1.001
% F198:10 % 800 0 0 160 0
% F198:15 % 0 0 0 160 0
DATA F199
% F199:0 % 959.9999 0 0 16 17
% F199:5 % 1 1 1 1 1.001
% F199:10 % 800 0 0 160 0
% F199:15 % 0 0 0 160 0
DATA F200
% F200:0 % 959.9999 0 0 16 17
% F200:5 % 1 1 1 1 1.001
% F200:10 % 800 0 0 160 0
% F200:15 % 0 0 0 160 0
DATA F201
% F201:0 % 959.9999 0 0 16 17
% F201:5 % 1 1 1 1 1.001
% F201:10 % 800 0 0 160 0
% F201:15 % 0 0 0 160 0
DATA F203
% F203:0 % 0 0 48 16 45
% F203:5 % 1.5 1 1.5 1 1
DATA F204
% F204:0 % 19000 0 0 16 0
% F204:5 % 1 1 1 1 1
% F204:10 % 15000 0 0 4000 0
% F204:15 % 0 0 0 4000 0
DATA F205
% F205:0 % 0 30 41 45 45
% F205:5 % 1.3 1.5 1 1 1
DATA F209
% F209:0 % 208 0 0 16 0
% F209:5 % 1 1 1 1 1
% F209:10 % 200 0 0 3 3
% F209:15 % 2 0 0 3 3
% F209:20 % 2 0
DATA F210
% F210:0 % 0 1 6 18 45
% F210:5 % 1 1 1 1 1
